// Core §3.8: SchemaVersion FIRST, initialized to the expected version
TYPE ST_CylinderParCfg :
STRUCT
    SchemaVersion : UINT := 1;
    MoveTimeout   : TIME := T#2S;
END_STRUCT
END_TYPE

(* stored: Version 1.1.0.1, ProductVersion 3.1.4024.12
   DUT ST_CylinderParCfg: Id {19a484f8-fe46-4cb6-a661-ff9a22a3cb34} *)
